FUNCTION_BLOCK XtsAxis
VAR_INPUT
END_VAR
VAR_OUTPUT
END_VAR
VAR

	Axis			: AXIS_REF;
	
	BusyMoving				: BOOL;
	BusyStopping			: BOOL;
	Error					: BOOL;
	ErrorID					: UDINT;
	ErrorIDPrevious			: UDINT;
	ErrorStop				: BOOL;
	Disabled				: BOOL;
	Stopping				: BOOL;
	StandStill				: BOOL;
	DiscreteMotion			: BOOL;
	ContinuousMotion		: BOOL;
	SynchronizedMotion		: BOOL;
	Homing					: BOOL;
	ConstantVelocity		: BOOL;
	Accelerating			: BOOL;
	Decelerating			: BOOL;
	Status					: ST_AxisStatus;
	ErrorCount				: UINT;

END_VAR

// NETWORK 1

END_FUNCTION_BLOCK

(* stored: Version 1.1.0.1, ProductVersion 3.1.4024.12
   POU XtsAxis: Id {ec1eec99-a289-419f-92b9-8b98742473d8}, SpecialFunc None
   Folder Movements: Id {e983c8f8-8927-4dc9-9aed-b49726e466f0}
   Folder Power and Utility: Id {27299485-0fb2-48d8-a5a9-eb5b18706a1b} *)
